FUNCTION_BLOCK TimeProvider
VAR_INPUT
END_VAR
VAR_OUTPUT
END_VAR
VAR
	localSystemTime						: FB_LocalSystemTime;
	
	// timestamp
	getTimeZoneInformation 			: FB_GetTimeZoneInformation;
    timeZoneInformation 			: ST_TimeZoneInformation;
    specificLocalTimeToFileTime 	: FB_TzSpecificLocalTimeToFileTime;
    fileTime						: T_FILETIME;
    onZerothSecondLastCycle 		: BOOL;
END_VAR

localSystemTime(bEnable := FALSE);


//https://stackoverflow.com/questions/41773732/how-do-i-get-the-unix-timestamp-in-twincat3

// On the zeroth second of each minutesync timezone information
IF (timeZoneInformation.standardName = '' OR (localSystemTime.systemTime.wSecond = 0 AND NOT onZerothSecondLastCycle)) THEN
    getTimeZoneInformation(sNetID := '', bExecute := TRUE, tzInfo => timeZoneInformation);
END_IF;

// Convert local system time to unix timestamps
specificLocalTimeToFileTime(in := Tc2_Utilities.SYSTEMTIME_TO_FILETIME(localSystemTime.systemTime), tzInfo := timeZoneInformation, out => fileTime);
//seconds := (SHL(DWORD_TO_ULINT(fileTime.dwHighDateTime), 32) + DWORD_TO_ULINT(fileTime.dwLowDateTime)) / 10000000 - 11644473600;
//milliseconds := (SHL(DWORD_TO_ULINT(fileTime.dwHighDateTime), 32) + DWORD_TO_ULINT(fileTime.dwLowDateTime)) / 10000 - 11644473600000;

onZerothSecondLastCycle := localSystemTime.systemTime.wSecond = 0;

METHOD FB_init : BOOL
VAR_INPUT
	bInitRetains : BOOL; // if TRUE, the retain variables are initialized (warm start / cold start)
	bInCopyCode : BOOL;  // if TRUE, the instance afterwards gets moved into the copy code (online change)
END_VAR
localSystemTime(bEnable := TRUE);
END_METHOD

METHOD GetMonthName : STRING
VAR_INPUT
	monthNumber			: UINT;
	shortName			: BOOL;
END_VAR
IF shortName THEN
	CASE monthNumber OF
		1	: GetMonthName := 'Jan';
		2	: GetMonthName := 'Feb';
		3	: GetMonthName := 'Mar';
		4	: GetMonthName := 'Apr';
		5	: GetMonthName := 'May';
		6	: GetMonthName := 'Jun';
		7	: GetMonthName := 'Jul';
		8	: GetMonthName := 'Aug';
		9	: GetMonthName := 'Sep';
		10	: GetMonthName := 'Oct';
		11	: GetMonthName := 'Nov';
		12	: GetMonthName := 'Dec';
	END_CASE
ELSE
	CASE monthNumber OF
		1	: GetMonthName := 'January';
		2	: GetMonthName := 'February';
		3	: GetMonthName := 'March';
		4	: GetMonthName := 'April';
		5	: GetMonthName := 'May';
		6	: GetMonthName := 'June';
		7	: GetMonthName := 'July';
		8	: GetMonthName := 'August';
		9	: GetMonthName := 'September';
		10	: GetMonthName := 'October';
		11	: GetMonthName := 'November';
		12	: GetMonthName := 'December';
	END_CASE
END_IF
END_METHOD

METHOD GetTimeString : STRING
VAR_INPUT
	format : STRING; //hh:mm:ss:SSS dd:MM:yyyy https://www.ibm.com/docs/en/rtw/9.0.1?topic=reference-formatting-parsing-date-time-patterns
END_VAR
VAR
	re : Regex;
END_VAR
// TODO: needs rework
(*
	regex - also can return matched string
	while re.length > 0
		case regex.string
			h
			hh
			m
			mm
			mmm
			.
			.
			.
*)


GetTimeString := format;

re.match('{hh*}', GetTimeString);
CASE re.length OF
	3 : 
		GetTimeString := REPLACE( STR1 := GetTimeString, STR2 := TO_STRING(localSystemTime.systemTime.wHour), L := re.length, P := re.start);
	4 :
		GetTimeString := REPLACE( STR1 := GetTimeString, STR2 := AddLeadingZeros(TO_STRING(localSystemTime.systemTime.wHour), 2), L := re.length, P := re.start);
END_CASE
re.match('{mm*}', GetTimeString);
CASE re.length OF
	3 : 
		GetTimeString := REPLACE( STR1 := GetTimeString, STR2 := TO_STRING(localSystemTime.systemTime.wMinute), L := re.length, P := re.start);
	4 :
		GetTimeString := REPLACE( STR1 := GetTimeString, STR2 := AddLeadingZeros(TO_STRING(localSystemTime.systemTime.wMinute), 2), L := re.length, P := re.start);
END_CASE
re.match('{ss*}', GetTimeString);
CASE re.length OF
	3 : 
		GetTimeString := REPLACE( STR1 := GetTimeString, STR2 := TO_STRING(localSystemTime.systemTime.wSecond), L := re.length, P := re.start);
	4 :
		GetTimeString := REPLACE( STR1 := GetTimeString, STR2 := AddLeadingZeros(TO_STRING(localSystemTime.systemTime.wSecond), 2), L := re.length, P := re.start);
END_CASE
re.match('{SS*}', GetTimeString);
CASE re.length OF
	3 : 
		GetTimeString := REPLACE( STR1 := GetTimeString, STR2 := TO_STRING(localSystemTime.systemTime.wMilliseconds/100), L := re.length, P := re.start);
	4 :
		GetTimeString := REPLACE( STR1 := GetTimeString, STR2 := AddLeadingZeros(TO_STRING(localSystemTime.systemTime.wMilliseconds/10), 2), L := re.length, P := re.start);
	5 :
		GetTimeString := REPLACE( STR1 := GetTimeString, STR2 := AddLeadingZeros(TO_STRING(localSystemTime.systemTime.wMilliseconds), 3), L := re.length, P := re.start);
END_CASE

re.match('{dd*}', GetTimeString);
CASE re.length OF
	3 : 
		GetTimeString := REPLACE( STR1 := GetTimeString, STR2 := TO_STRING(localSystemTime.systemTime.wDay), L := re.length, P := re.start);
	4 :
		GetTimeString := REPLACE( STR1 := GetTimeString, STR2 := AddLeadingZeros(TO_STRING(localSystemTime.systemTime.wDay), 2), L := re.length, P := re.start);
	5:
		GetTimeString := REPLACE( STR1 := GetTimeString, STR2 := GetWeekdayName(localSystemTime.systemTime.wDayOfWeek, TRUE), L := re.length, P := re.start);
	6:
		GetTimeString := REPLACE( STR1 := GetTimeString, STR2 := GetWeekdayName(localSystemTime.systemTime.wDayOfWeek, FALSE), L := re.length, P := re.start);
END_CASE
re.match('{MM*}', GetTimeString);
CASE re.length OF
	3 : 
		GetTimeString := REPLACE( STR1 := GetTimeString, STR2 := TO_STRING(localSystemTime.systemTime.wMonth), L := re.length, P := re.start);
	4 :
		GetTimeString := REPLACE( STR1 := GetTimeString, STR2 := AddLeadingZeros(TO_STRING(localSystemTime.systemTime.wMonth), 2), L := re.length, P := re.start);
	5:
		GetTimeString := REPLACE( STR1 := GetTimeString, STR2 := GetMonthName(localSystemTime.systemTime.wMonth, TRUE), L := re.length, P := re.start);
	6:
		GetTimeString := REPLACE( STR1 := GetTimeString, STR2 := GetMonthName(localSystemTime.systemTime.wMonth, FALSE), L := re.length, P := re.start);
END_CASE
re.match('{yy*}', GetTimeString);
CASE re.length OF
	3..6 : 
		GetTimeString := REPLACE( STR1 := GetTimeString, STR2 := RIGHT(TO_STRING(localSystemTime.systemTime.wYear), re.length - 2), L := re.length, P := re.start);
END_CASE
END_METHOD

METHOD GetWeekdayName : STRING
VAR_INPUT
	weekDayNumber		: UINT;
	shortName			: BOOL;
END_VAR
IF shortName THEN
	CASE weekDayNumber OF
		0	: GetWeekdayName := 'Sun';
		1	: GetWeekdayName := 'Mon';
		2	: GetWeekdayName := 'Tue';
		3	: GetWeekdayName := 'Wed';
		4	: GetWeekdayName := 'Thu';
		5	: GetWeekdayName := 'Fri';
		6	: GetWeekdayName := 'Sat';
	END_CASE
ELSE
	CASE weekDayNumber OF
		0	: GetWeekdayName := 'Sunday';
		1	: GetWeekdayName := 'Monday';
		2	: GetWeekdayName := 'Tuesday';
		3	: GetWeekdayName := 'Wednesday';
		4	: GetWeekdayName := 'Thursday';
		5	: GetWeekdayName := 'Friday';
		6	: GetWeekdayName := 'Saturday';
	END_CASE
END_IF
END_METHOD

PROPERTY Timestamp : ULINT // Unix timestamp in milliseconds
GET
// TODO is this even right?
Timestamp := (SHL(DWORD_TO_ULINT(fileTime.dwHighDateTime), 32) + DWORD_TO_ULINT(fileTime.dwLowDateTime)) / 10000 - 11644473600000;
END_GET
END_PROPERTY

PROPERTY TimeStruct : TIMESTRUCT // Week starts with Sunday
GET
TimeStruct := localSystemTime.systemTime;
END_GET
END_PROPERTY

PROPERTY TimeStructISO8601 : TIMESTRUCT // Week starts with Monday
GET
TimeStructISO8601 := localSystemTime.systemTime;
IF TimeStructISO8601.wDayOfWeek = 0 THEN
	TimeStructISO8601.wDayOfWeek := 6; // Move Sunday to the end of the week
ELSE
	TimeStructISO8601.wDayOfWeek := TimeStructISO8601.wDayOfWeek - 1;
END_IF
END_GET
END_PROPERTY

END_FUNCTION_BLOCK

(* stored: Version 1.1.0.1, ProductVersion 3.1.4024.11
   POU TimeProvider: Id {e0628be4-a9c9-48e0-bed6-4aecca528c6a}, SpecialFunc None
   Method FB_init: Id {0eeee39d-a42c-4906-b99a-b1a54180bb7e}
   Method GetMonthName: Id {91d99de0-20f1-48c5-955c-7131500af3fe}
   Method GetTimeString: Id {679679f2-ee04-47f6-8dbf-036ccba99ed1}
   Method GetWeekdayName: Id {99a7f3ff-bde0-440a-b816-7ab555a7320b}
   Property Timestamp: Id {08bcd9a2-bdae-4771-98e3-9c00ad89897d}
   Get Get: Id {e69d997d-74c0-42cf-885a-62d0470c50b9}
   Property TimeStruct: Id {297e10ee-4ad8-4580-817a-d120a347bf4a}
   Get Get: Id {a9eb649c-2014-4f19-aa8e-497503863d4e}
   Property TimeStructISO8601: Id {ac78a099-70e2-4548-bf43-8738b34279ec}
   Get Get: Id {d91c40a9-9619-4d0f-86b9-f7b899b22f54} *)
